INTERFACE I_SignalHandling

METHOD BuildSignal : ST_Signal
VAR_INPUT
	eSignal	: E_Signal;
END_VAR
END_METHOD

METHOD GenericReceive : BOOL
VAR_INPUT
	eSignal : E_Signal;
END_VAR
END_METHOD

PROPERTY getSignal : ST_Signal
GET
END_GET
END_PROPERTY

PROPERTY getSignalOrigin : E_Origin
GET
END_GET
END_PROPERTY

METHOD GlobalReset 
VAR_INPUT
END_VAR
END_METHOD

METHOD Receive : BOOL
VAR_INPUT
	eSignal : E_Signal;
	eSignalOrigin : E_Origin;
END_VAR
END_METHOD

METHOD ResetSignal : BOOL
VAR_INPUT
	eSignal : E_Signal;
	eSignalOrigin : E_Origin;
END_VAR
END_METHOD

METHOD Signal : BOOL
VAR_INPUT
	stSignal	: ST_Signal;
END_VAR
END_METHOD

METHOD SignalAvailable : BOOL
VAR_INPUT
END_VAR
END_METHOD

END_INTERFACE

(* stored: Version 1.1.0.1, ProductVersion 3.1.4024.0
   Itf I_SignalHandling: Id {722a65b6-464f-4fbf-a750-56f3314823ba}
   Method BuildSignal: Id {33a22f54-49cb-472f-a974-18d053e92171}
   Method GenericReceive: Id {e3082482-868e-4e97-82aa-e6e8309b155b}
   Property getSignal: Id {f5c45975-da8b-449d-8570-cf3ec81259bf}
   Get Get: Id {8b0e9c41-5f27-402e-92bd-9fe90333feab}
   Property getSignalOrigin: Id {1ef738a6-05a6-4e72-bd7a-fc777537a3c4}
   Get Get: Id {29bcce1f-f953-440a-8a05-78fd4f7b0260}
   Method GlobalReset: Id {21e98d47-dcd8-4290-9f78-f6060bc68a95}
   Method Receive: Id {059b0042-9096-44c1-9b92-dc16887c27ee}
   Method ResetSignal: Id {ccea8a91-62d7-4493-9a0a-5a00360cd0ce}
   Method Signal: Id {164a721d-6a00-4434-ab87-0692cba2a478}
   Method SignalAvailable: Id {1576c7ba-0127-42b8-aecf-634dd8d6a0f2} *)
